TYPE "tFullSignalInt"
VERSION : 0.8
   STRUCT
      scale : "tScale";
      i : Int;
      signal : Int;
   END_STRUCT;

END_TYPE

